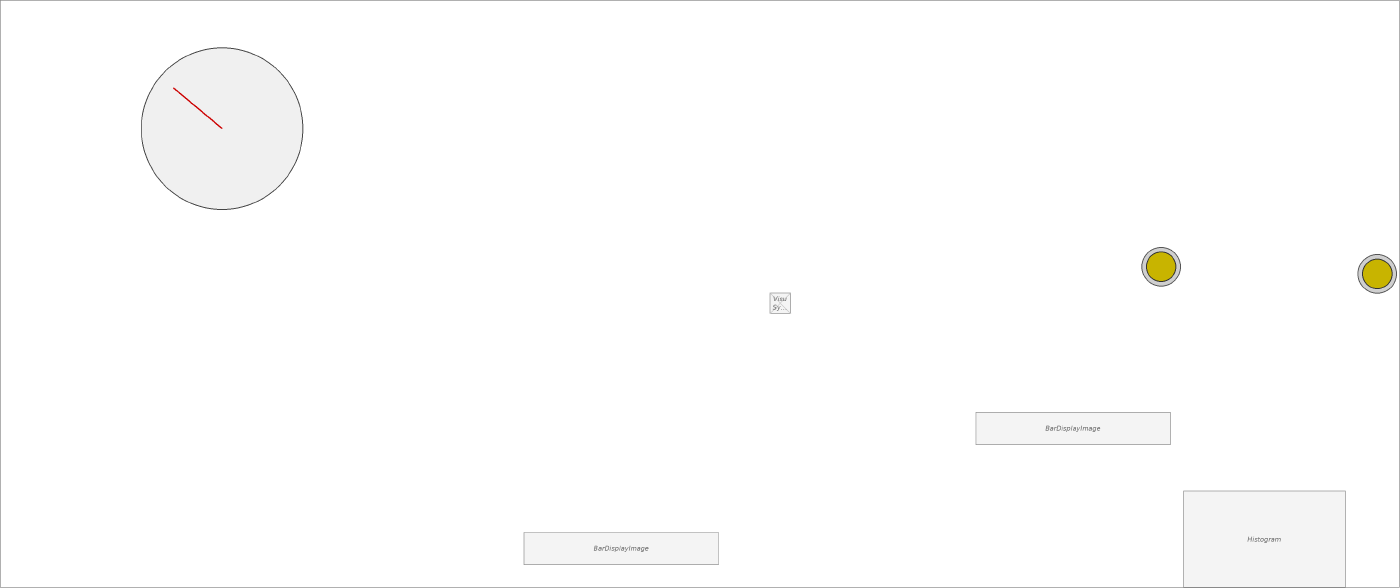
VISUALIZATION Visualization  // 2157x906
    Lamp1 (2087,387 70x70), style: Lamp-Lamp1-Yellow
    Lamp1 (1754,376 70x70), variable: Inputs.DI_HOISTING_LIM_TOP, style: Lamp-Lamp1-Yellow
    Meter360 (217,73 250x250), value: Inputs.AI_PressureSensor, style: Meter-Meter360-Gray, scale format: %.1f, scale 0..100
    BarDisplayImage (807,820 300x50), value: Process.Pressure, style: BarDisplayImage-Gray, scale format: %.1f, scale 0..100
    Histogram (1823,756 250x150), scale format: %.1f, scale 0..100
    BarDisplayImage (1503,635 300x50), value: Process.Temperature, style: BarDisplayImage-Gray, scale format: %.1f, scale 0..100
    Image (1186,451 32x32), text variable: Process.Temperature, image: VisuSymbols.Symbols.Text
END_VISUALIZATION

(* stored: Version 1.1.0.1, ProductVersion 3.1.4024.9
   Visu Visualization: Id {848a49a0-95b9-44c1-9e64-949fccc00c1f} *)
